// TIA Portal V19 export
FUNCTION "Area01_HU_CALL" : Void   // FC128, LAD
TITLE = COIL HANDLING MAIN HU (7,5kW) CALL
// stored: SetENOAutomatically false
   VAR_TEMP
      retval : Int;
      OilTemperature : Real;
      AnalTemperature_Real : Real;
   END_VAR
BEGIN

REGION Network 1: Machine Manager
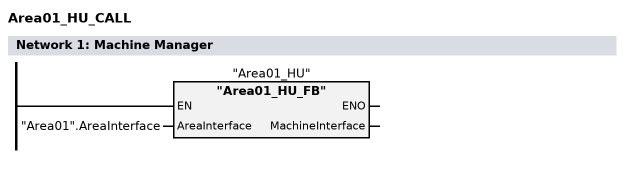
   RUNG wire#powerrail
      "Area01_HU"(AreaInterface := "Area01".AreaInterface, MachineInterface =>)
   END_RUNG
   // the same network as SCL:
   "Area01_HU"(AreaInterface := "Area01".AreaInterface);   // "Area01_HU_FB"
END_REGION
END_FUNCTION
